{attribute 'qualified_only'}
VAR_GLOBAL
END_VAR

(* stored: Version 1.1.0.1, ProductVersion 3.1.4024.9
   GVL GVL_1: Id {244adde5-a0e4-4d27-beed-468ac67dddcc} *)
